// TIA Portal V17 export
// export: Created 2025-05-22T06:02:00.7232443Z, ExportSetting WithDefaults, DisplayName Totally Integrated Automation Portal, DisplayVersion V17 Update 8, DisplayName TIA Portal Openness, DisplayVersion V17 Update 8, DisplayName TIA Portal Version Control Interface, DisplayVersion V17, DisplayName SINAMICS Startdrive Advanced, DisplayVersion V17 SP2, DisplayName SINAMICS Startdrive G110M, G120, G120C, G120D, G120P, G115D, DisplayVersion V17 SP2, DisplayName SINAMICS Startdrive G130, G150, S120, S150, SINAMICS MV, S210, DisplayVersion V17 SP2, DisplayName STEP 7 Professional, DisplayVersion V17 Update 8, DisplayName SINUMERIK ONE STEP 7 Toolbox, DisplayVersion V17 Update 12, DisplayName SINUMERIK ONE PLC Basic Program Plus, DisplayVersion V17 Update 12, DisplayName SINUMERIK 840D sl STEP 7 Toolbox, DisplayVersion V17 Update 12, DisplayName STEP 7 Safety, DisplayVersion V17 Update 6, DisplayName WinCC Advanced, DisplayVersion V17 Update 8
FUNCTION "FC17900_MAINTENANCE_SEQUENCE" : Void   // FC17001, LAD
{ S7_Optimized_Access := 'TRUE' }
VERSION : 0.1
// stored: AutoNumber false, IsIECCheckEnabled false, SetENOAutomatically false, UDAEnableTagReadback false
   VAR_INPUT
      START_REQ : Bool;
      NUMBER_STEPS : Int;
      FIRST_STEP_DONE : Bool;
      SECOND_STEP_DONE : Bool;
      THRID_STEP_DONE : Bool;
      FOURTH_STEP_DONE : Bool;
      FIFTH_STEP_DONE : Bool;
   END_VAR
   VAR_OUTPUT
      FIRST_OPERATOR_HELP : Bool;
      SECOND_OPERATOR_HELP : Bool;
      THRID_OPERATOR_HELP : Bool;
      FOURTH_OPERATOR_HELP : Bool;
      FIFTH_OPERATOR_HELP : Bool;
      MAINTENANCE_IN_PROGRESS : Bool;
   END_VAR
   VAR_TEMP
      OPTION_FIRST_STEP : Bool;
      OPTION_SECOND_STEP : Bool;
      OPTION_THRID_STEP : Bool;
      OPTION_FOURTH_STEP : Bool;
      OPTION_FIFTH_STEP : Bool;
      SEQUENCE : "SEQUENCE";
   END_VAR
   VAR_TEMP   // added for the SCL form of the ladder/FBD networks
      _w1 : Bool;
   END_VAR
BEGIN

REGION Network 1: RESET OPTIONS
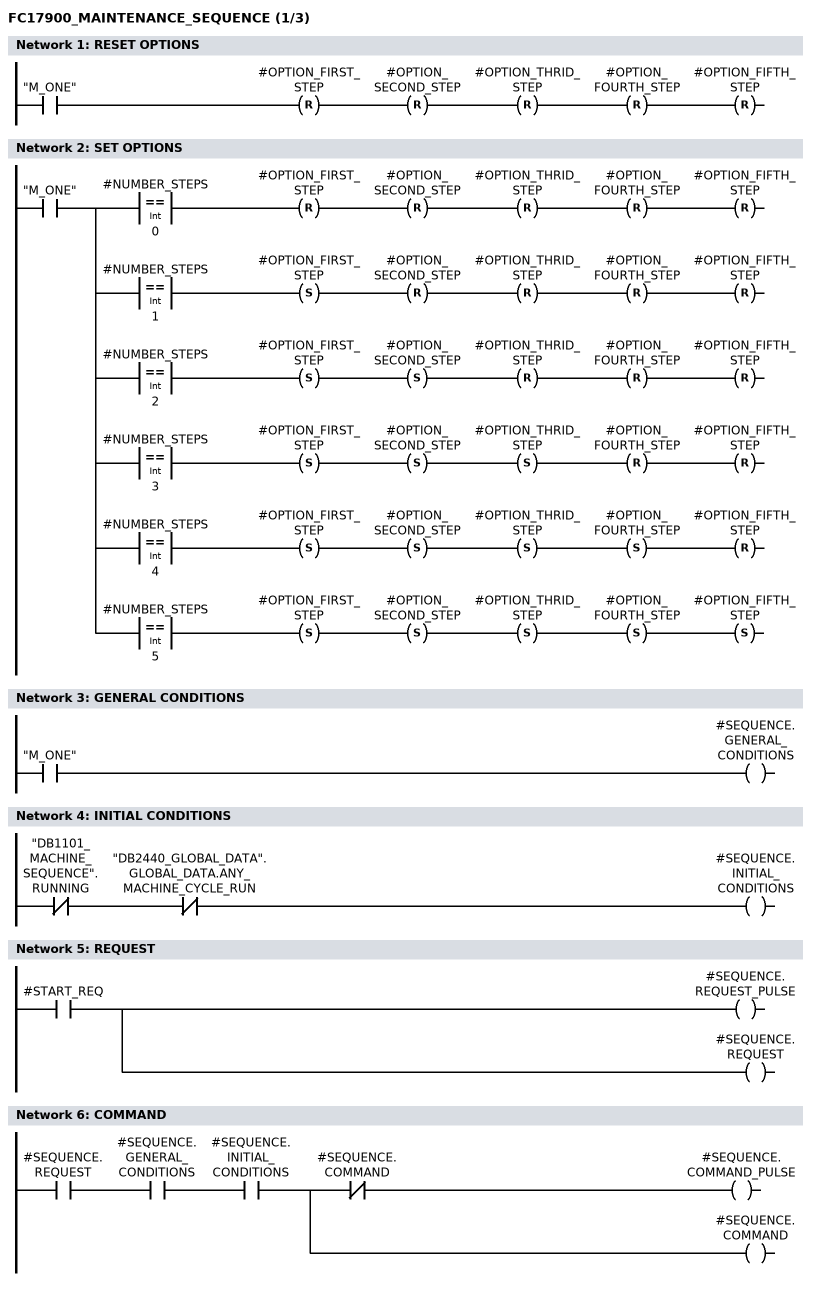
   RUNG wire#powerrail
      Contact( "M_ONE" )
      R_Coil( #OPTION_FIRST_STEP )
      R_Coil( #OPTION_SECOND_STEP )
      R_Coil( #OPTION_THRID_STEP )
      R_Coil( #OPTION_FOURTH_STEP )
      R_Coil( #OPTION_FIFTH_STEP )
   END_RUNG
   // the same network as SCL:
   IF "M_ONE" THEN
       #OPTION_FIRST_STEP := FALSE;
       #OPTION_SECOND_STEP := FALSE;
       #OPTION_THRID_STEP := FALSE;
       #OPTION_FOURTH_STEP := FALSE;
       #OPTION_FIFTH_STEP := FALSE;
   END_IF;
END_REGION

REGION Network 2: SET OPTIONS
   RUNG wire#powerrail
      Contact( "M_ONE" )
      wire#w1
      { S7_Templates := "SrcType := Int" } EQ_Contact(in1 := #NUMBER_STEPS, in2 := 0)
      R_Coil( #OPTION_FIRST_STEP )
      R_Coil( #OPTION_SECOND_STEP )
      R_Coil( #OPTION_THRID_STEP )
      R_Coil( #OPTION_FOURTH_STEP )
      R_Coil( #OPTION_FIFTH_STEP )
   END_RUNG
   RUNG wire#w1
      { S7_Templates := "SrcType := Int" } EQ_Contact(in1 := #NUMBER_STEPS, in2 := 1)
      S_Coil( #OPTION_FIRST_STEP )
      R_Coil( #OPTION_SECOND_STEP )
      R_Coil( #OPTION_THRID_STEP )
      R_Coil( #OPTION_FOURTH_STEP )
      R_Coil( #OPTION_FIFTH_STEP )
   END_RUNG
   RUNG wire#w1
      { S7_Templates := "SrcType := Int" } EQ_Contact(in1 := #NUMBER_STEPS, in2 := 2)
      S_Coil( #OPTION_FIRST_STEP )
      S_Coil( #OPTION_SECOND_STEP )
      R_Coil( #OPTION_THRID_STEP )
      R_Coil( #OPTION_FOURTH_STEP )
      R_Coil( #OPTION_FIFTH_STEP )
   END_RUNG
   RUNG wire#w1
      { S7_Templates := "SrcType := Int" } EQ_Contact(in1 := #NUMBER_STEPS, in2 := 3)
      S_Coil( #OPTION_FIRST_STEP )
      S_Coil( #OPTION_SECOND_STEP )
      S_Coil( #OPTION_THRID_STEP )
      R_Coil( #OPTION_FOURTH_STEP )
      R_Coil( #OPTION_FIFTH_STEP )
   END_RUNG
   RUNG wire#w1
      { S7_Templates := "SrcType := Int" } EQ_Contact(in1 := #NUMBER_STEPS, in2 := 4)
      S_Coil( #OPTION_FIRST_STEP )
      S_Coil( #OPTION_SECOND_STEP )
      S_Coil( #OPTION_THRID_STEP )
      S_Coil( #OPTION_FOURTH_STEP )
      R_Coil( #OPTION_FIFTH_STEP )
   END_RUNG
   RUNG wire#w1
      { S7_Templates := "SrcType := Int" } EQ_Contact(in1 := #NUMBER_STEPS, in2 := 5)
      S_Coil( #OPTION_FIRST_STEP )
      S_Coil( #OPTION_SECOND_STEP )
      S_Coil( #OPTION_THRID_STEP )
      S_Coil( #OPTION_FOURTH_STEP )
      S_Coil( #OPTION_FIFTH_STEP )
   END_RUNG
   // the same network as SCL:
   IF "M_ONE" AND (#NUMBER_STEPS = 0) THEN
       #OPTION_FIRST_STEP := FALSE;
       #OPTION_SECOND_STEP := FALSE;
       #OPTION_THRID_STEP := FALSE;
       #OPTION_FOURTH_STEP := FALSE;
       #OPTION_FIFTH_STEP := FALSE;
   END_IF;
   IF "M_ONE" AND (#NUMBER_STEPS = 1) THEN
       #OPTION_FIRST_STEP := TRUE;
       #OPTION_SECOND_STEP := FALSE;
       #OPTION_THRID_STEP := FALSE;
       #OPTION_FOURTH_STEP := FALSE;
       #OPTION_FIFTH_STEP := FALSE;
   END_IF;
   IF "M_ONE" AND (#NUMBER_STEPS = 2) THEN
       #OPTION_FIRST_STEP := TRUE;
       #OPTION_SECOND_STEP := TRUE;
       #OPTION_THRID_STEP := FALSE;
       #OPTION_FOURTH_STEP := FALSE;
       #OPTION_FIFTH_STEP := FALSE;
   END_IF;
   IF "M_ONE" AND (#NUMBER_STEPS = 3) THEN
       #OPTION_FIRST_STEP := TRUE;
       #OPTION_SECOND_STEP := TRUE;
       #OPTION_THRID_STEP := TRUE;
       #OPTION_FOURTH_STEP := FALSE;
       #OPTION_FIFTH_STEP := FALSE;
   END_IF;
   IF "M_ONE" AND (#NUMBER_STEPS = 4) THEN
       #OPTION_FIRST_STEP := TRUE;
       #OPTION_SECOND_STEP := TRUE;
       #OPTION_THRID_STEP := TRUE;
       #OPTION_FOURTH_STEP := TRUE;
       #OPTION_FIFTH_STEP := FALSE;
   END_IF;
   IF "M_ONE" AND (#NUMBER_STEPS = 5) THEN
       #OPTION_FIRST_STEP := TRUE;
       #OPTION_SECOND_STEP := TRUE;
       #OPTION_THRID_STEP := TRUE;
       #OPTION_FOURTH_STEP := TRUE;
       #OPTION_FIFTH_STEP := TRUE;
   END_IF;
END_REGION

REGION Network 3: GENERAL CONDITIONS
   RUNG wire#powerrail
      Contact( "M_ONE" )
      Coil( #SEQUENCE.GENERAL_CONDITIONS )
   END_RUNG
   // the same network as SCL:
   #SEQUENCE.GENERAL_CONDITIONS := "M_ONE";
END_REGION

REGION Network 4: INITIAL CONDITIONS
   RUNG wire#powerrail
      I_Contact( "DB1101_MACHINE_SEQUENCE".RUNNING )
      I_Contact( "DB2440_GLOBAL_DATA".GLOBAL_DATA.ANY_MACHINE_CYCLE_RUN )
      Coil( #SEQUENCE.INITIAL_CONDITIONS )
   END_RUNG
   // the same network as SCL:
   #SEQUENCE.INITIAL_CONDITIONS := NOT "DB1101_MACHINE_SEQUENCE".RUNNING AND NOT "DB2440_GLOBAL_DATA".GLOBAL_DATA.ANY_MACHINE_CYCLE_RUN;
END_REGION

REGION Network 5: REQUEST
   RUNG wire#powerrail
      Contact( #START_REQ )
      wire#w1
      Coil( #SEQUENCE.REQUEST_PULSE )
   END_RUNG
   RUNG wire#w1
      Coil( #SEQUENCE.REQUEST )
   END_RUNG
   // the same network as SCL:
   #SEQUENCE.REQUEST_PULSE := #START_REQ;
   #SEQUENCE.REQUEST := #START_REQ;
END_REGION

REGION Network 6: COMMAND
   RUNG wire#powerrail
      Contact( #SEQUENCE.REQUEST )
      Contact( #SEQUENCE.GENERAL_CONDITIONS )
      Contact( #SEQUENCE.INITIAL_CONDITIONS )
      wire#w1
      I_Contact( #SEQUENCE.COMMAND )
      Coil( #SEQUENCE.COMMAND_PULSE )
   END_RUNG
   RUNG wire#w1
      Coil( #SEQUENCE.COMMAND )
   END_RUNG
   // the same network as SCL:
   #_w1 := #SEQUENCE.REQUEST AND #SEQUENCE.GENERAL_CONDITIONS AND #SEQUENCE.INITIAL_CONDITIONS;
   #SEQUENCE.COMMAND_PULSE := #_w1 AND NOT #SEQUENCE.COMMAND;
   #SEQUENCE.COMMAND := #_w1;
END_REGION

REGION Network 7: RESET PLC AND CNC
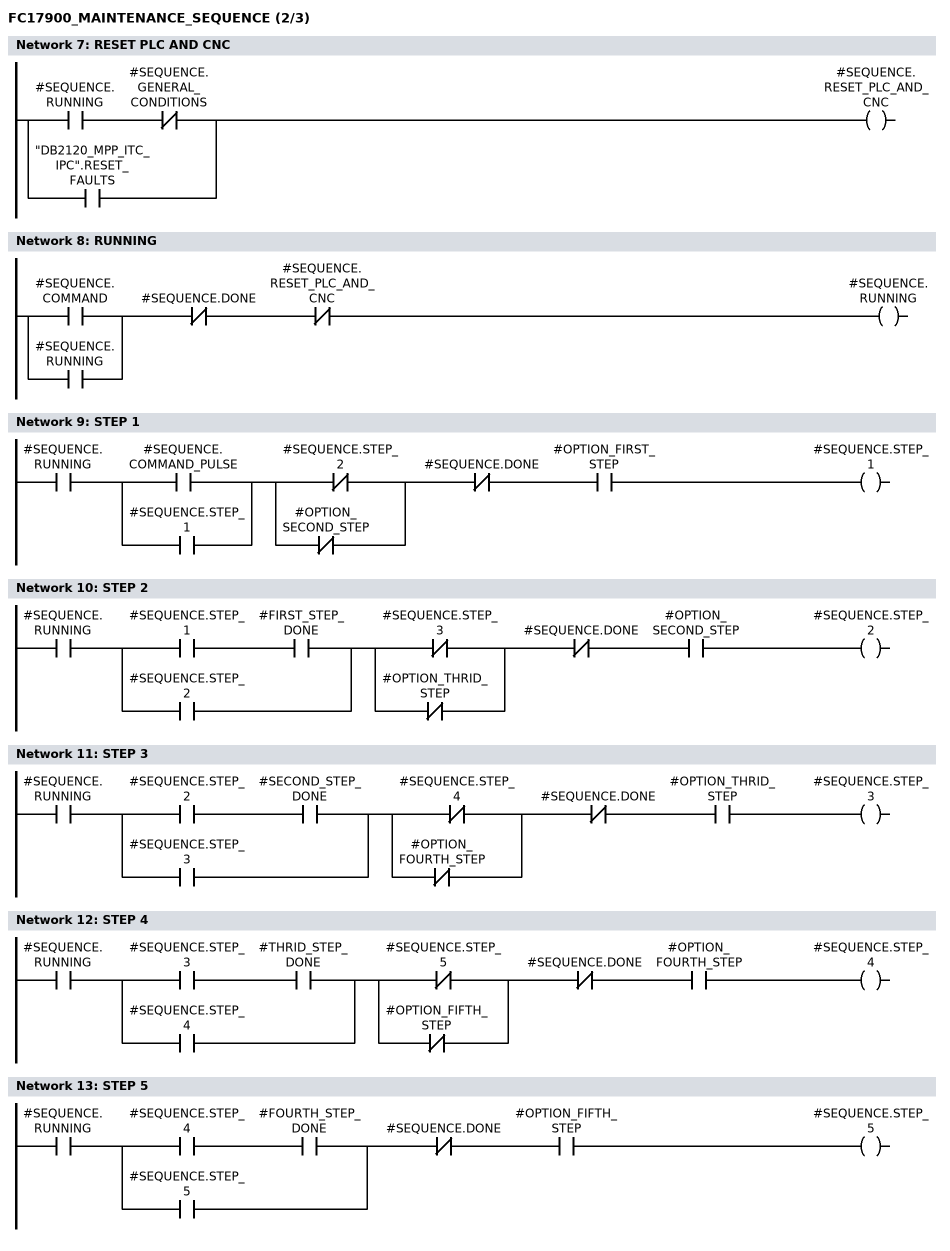
   RUNG wire#powerrail
      Contact( #SEQUENCE.RUNNING )
      I_Contact( #SEQUENCE.GENERAL_CONDITIONS )
      wire#w1
      Coil( #SEQUENCE.RESET_PLC_AND_CNC )
   END_RUNG
   RUNG wire#powerrail
      Contact( "DB2120_MPP_ITC_IPC".RESET_FAULTS )
   END_RUNG wire#w1
   // the same network as SCL:
   #SEQUENCE.RESET_PLC_AND_CNC := (#SEQUENCE.RUNNING AND NOT #SEQUENCE.GENERAL_CONDITIONS) OR "DB2120_MPP_ITC_IPC".RESET_FAULTS;
END_REGION

REGION Network 8: RUNNING
   RUNG wire#powerrail
      Contact( #SEQUENCE.COMMAND )
      wire#w1
      I_Contact( #SEQUENCE.DONE )
      I_Contact( #SEQUENCE.RESET_PLC_AND_CNC )
      Coil( #SEQUENCE.RUNNING )
   END_RUNG
   RUNG wire#powerrail
      Contact( #SEQUENCE.RUNNING )
   END_RUNG wire#w1
   // the same network as SCL:
   #SEQUENCE.RUNNING := (#SEQUENCE.COMMAND OR #SEQUENCE.RUNNING) AND NOT #SEQUENCE.DONE AND NOT #SEQUENCE.RESET_PLC_AND_CNC;
END_REGION

REGION Network 9: STEP 1
   RUNG wire#powerrail
      Contact( #SEQUENCE.RUNNING )
      wire#w1
      Contact( #SEQUENCE.COMMAND_PULSE )
      wire#w2
      I_Contact( #SEQUENCE.STEP_2 )
      wire#w3
      I_Contact( #SEQUENCE.DONE )
      Contact( #OPTION_FIRST_STEP )
      Coil( #SEQUENCE.STEP_1 )
   END_RUNG
   RUNG wire#w1
      Contact( #SEQUENCE.STEP_1 )
   END_RUNG wire#w2
   RUNG wire#w2
      I_Contact( #OPTION_SECOND_STEP )
   END_RUNG wire#w3
   // the same network as SCL:
   #SEQUENCE.STEP_1 := #SEQUENCE.RUNNING AND (#SEQUENCE.COMMAND_PULSE OR #SEQUENCE.STEP_1) AND (NOT #SEQUENCE.STEP_2 OR NOT #OPTION_SECOND_STEP) AND NOT #SEQUENCE.DONE AND #OPTION_FIRST_STEP;
END_REGION

REGION Network 10: STEP 2
   RUNG wire#powerrail
      Contact( #SEQUENCE.RUNNING )
      wire#w1
      Contact( #SEQUENCE.STEP_1 )
      Contact( #FIRST_STEP_DONE )
      wire#w2
      I_Contact( #SEQUENCE.STEP_3 )
      wire#w3
      I_Contact( #SEQUENCE.DONE )
      Contact( #OPTION_SECOND_STEP )
      Coil( #SEQUENCE.STEP_2 )
   END_RUNG
   RUNG wire#w1
      Contact( #SEQUENCE.STEP_2 )
   END_RUNG wire#w2
   RUNG wire#w2
      I_Contact( #OPTION_THRID_STEP )
   END_RUNG wire#w3
   // the same network as SCL:
   #SEQUENCE.STEP_2 := #SEQUENCE.RUNNING AND ((#SEQUENCE.STEP_1 AND #FIRST_STEP_DONE) OR #SEQUENCE.STEP_2) AND (NOT #SEQUENCE.STEP_3 OR NOT #OPTION_THRID_STEP) AND NOT #SEQUENCE.DONE AND #OPTION_SECOND_STEP;
END_REGION

REGION Network 11: STEP 3
   RUNG wire#powerrail
      Contact( #SEQUENCE.RUNNING )
      wire#w1
      Contact( #SEQUENCE.STEP_2 )
      Contact( #SECOND_STEP_DONE )
      wire#w2
      I_Contact( #SEQUENCE.STEP_4 )
      wire#w3
      I_Contact( #SEQUENCE.DONE )
      Contact( #OPTION_THRID_STEP )
      Coil( #SEQUENCE.STEP_3 )
   END_RUNG
   RUNG wire#w1
      Contact( #SEQUENCE.STEP_3 )
   END_RUNG wire#w2
   RUNG wire#w2
      I_Contact( #OPTION_FOURTH_STEP )
   END_RUNG wire#w3
   // the same network as SCL:
   #SEQUENCE.STEP_3 := #SEQUENCE.RUNNING AND ((#SEQUENCE.STEP_2 AND #SECOND_STEP_DONE) OR #SEQUENCE.STEP_3) AND (NOT #SEQUENCE.STEP_4 OR NOT #OPTION_FOURTH_STEP) AND NOT #SEQUENCE.DONE AND #OPTION_THRID_STEP;
END_REGION

REGION Network 12: STEP 4
   RUNG wire#powerrail
      Contact( #SEQUENCE.RUNNING )
      wire#w1
      Contact( #SEQUENCE.STEP_3 )
      Contact( #THRID_STEP_DONE )
      wire#w2
      I_Contact( #SEQUENCE.STEP_5 )
      wire#w3
      I_Contact( #SEQUENCE.DONE )
      Contact( #OPTION_FOURTH_STEP )
      Coil( #SEQUENCE.STEP_4 )
   END_RUNG
   RUNG wire#w1
      Contact( #SEQUENCE.STEP_4 )
   END_RUNG wire#w2
   RUNG wire#w2
      I_Contact( #OPTION_FIFTH_STEP )
   END_RUNG wire#w3
   // the same network as SCL:
   #SEQUENCE.STEP_4 := #SEQUENCE.RUNNING AND ((#SEQUENCE.STEP_3 AND #THRID_STEP_DONE) OR #SEQUENCE.STEP_4) AND (NOT #SEQUENCE.STEP_5 OR NOT #OPTION_FIFTH_STEP) AND NOT #SEQUENCE.DONE AND #OPTION_FOURTH_STEP;
END_REGION

REGION Network 13: STEP 5
   RUNG wire#powerrail
      Contact( #SEQUENCE.RUNNING )
      wire#w1
      Contact( #SEQUENCE.STEP_4 )
      Contact( #FOURTH_STEP_DONE )
      wire#w2
      I_Contact( #SEQUENCE.DONE )
      Contact( #OPTION_FIFTH_STEP )
      Coil( #SEQUENCE.STEP_5 )
   END_RUNG
   RUNG wire#w1
      Contact( #SEQUENCE.STEP_5 )
   END_RUNG wire#w2
   // the same network as SCL:
   #SEQUENCE.STEP_5 := #SEQUENCE.RUNNING AND ((#SEQUENCE.STEP_4 AND #FOURTH_STEP_DONE) OR #SEQUENCE.STEP_5) AND NOT #SEQUENCE.DONE AND #OPTION_FIFTH_STEP;
END_REGION

REGION Network 14: DONE
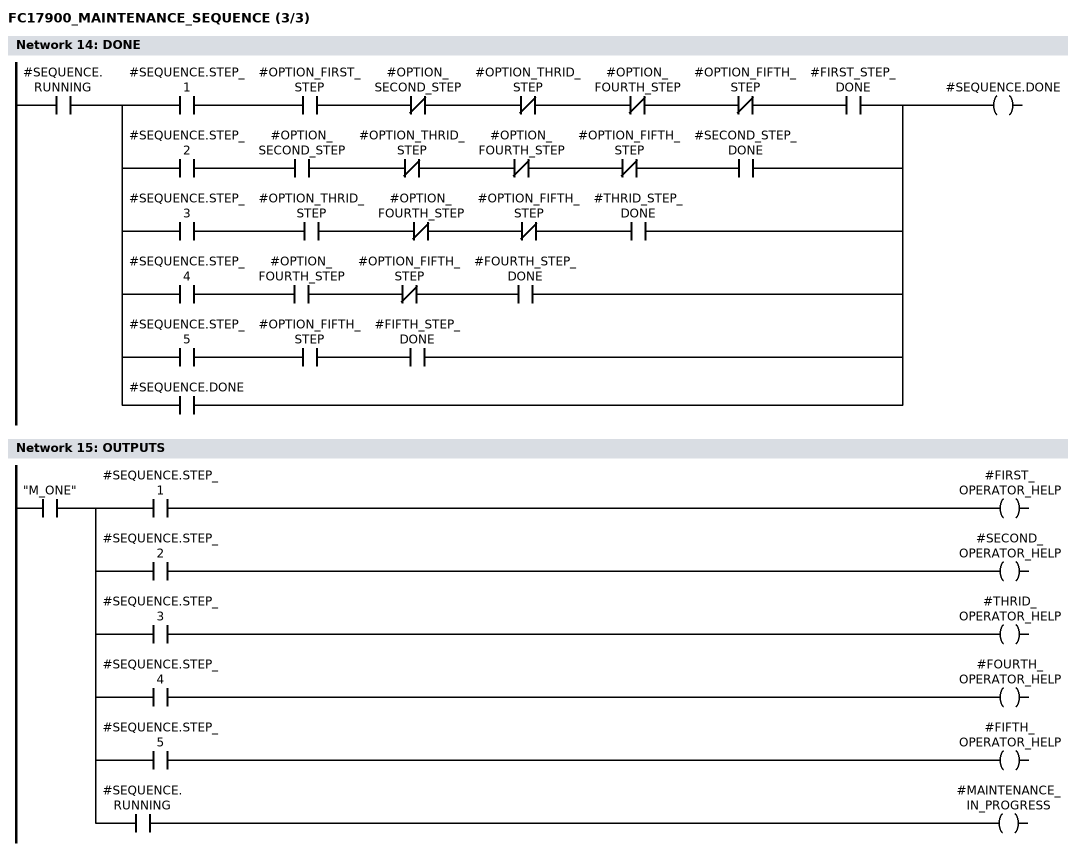
   RUNG wire#powerrail
      Contact( #SEQUENCE.RUNNING )
      wire#w1
      Contact( #SEQUENCE.STEP_1 )
      Contact( #OPTION_FIRST_STEP )
      I_Contact( #OPTION_SECOND_STEP )
      I_Contact( #OPTION_THRID_STEP )
      I_Contact( #OPTION_FOURTH_STEP )
      I_Contact( #OPTION_FIFTH_STEP )
      Contact( #FIRST_STEP_DONE )
      wire#w2
      Coil( #SEQUENCE.DONE )
   END_RUNG
   RUNG wire#w1
      Contact( #SEQUENCE.STEP_2 )
      Contact( #OPTION_SECOND_STEP )
      I_Contact( #OPTION_THRID_STEP )
      I_Contact( #OPTION_FOURTH_STEP )
      I_Contact( #OPTION_FIFTH_STEP )
      Contact( #SECOND_STEP_DONE )
   END_RUNG wire#w2
   RUNG wire#w1
      Contact( #SEQUENCE.STEP_3 )
      Contact( #OPTION_THRID_STEP )
      I_Contact( #OPTION_FOURTH_STEP )
      I_Contact( #OPTION_FIFTH_STEP )
      Contact( #THRID_STEP_DONE )
   END_RUNG wire#w2
   RUNG wire#w1
      Contact( #SEQUENCE.STEP_4 )
      Contact( #OPTION_FOURTH_STEP )
      I_Contact( #OPTION_FIFTH_STEP )
      Contact( #FOURTH_STEP_DONE )
   END_RUNG wire#w2
   RUNG wire#w1
      Contact( #SEQUENCE.STEP_5 )
      Contact( #OPTION_FIFTH_STEP )
      Contact( #FIFTH_STEP_DONE )
   END_RUNG wire#w2
   RUNG wire#w1
      Contact( #SEQUENCE.DONE )
   END_RUNG wire#w2
   // the same network as SCL:
   #SEQUENCE.DONE := #SEQUENCE.RUNNING AND ((#SEQUENCE.STEP_1 AND #OPTION_FIRST_STEP AND NOT #OPTION_SECOND_STEP AND NOT #OPTION_THRID_STEP AND NOT #OPTION_FOURTH_STEP AND NOT #OPTION_FIFTH_STEP AND #FIRST_STEP_DONE) OR (#SEQUENCE.STEP_2 AND #OPTION_SECOND_STEP AND NOT #OPTION_THRID_STEP AND NOT #OPTION_FOURTH_STEP AND NOT #OPTION_FIFTH_STEP AND #SECOND_STEP_DONE) OR (#SEQUENCE.STEP_3 AND #OPTION_THRID_STEP AND NOT #OPTION_FOURTH_STEP AND NOT #OPTION_FIFTH_STEP AND #THRID_STEP_DONE) OR (#SEQUENCE.STEP_4 AND #OPTION_FOURTH_STEP AND NOT #OPTION_FIFTH_STEP AND #FOURTH_STEP_DONE) OR (#SEQUENCE.STEP_5 AND #OPTION_FIFTH_STEP AND #FIFTH_STEP_DONE) OR #SEQUENCE.DONE);
END_REGION

REGION Network 15: OUTPUTS
   RUNG wire#powerrail
      Contact( "M_ONE" )
      wire#w1
      Contact( #SEQUENCE.STEP_1 )
      Coil( #FIRST_OPERATOR_HELP )
   END_RUNG
   RUNG wire#w1
      Contact( #SEQUENCE.STEP_2 )
      Coil( #SECOND_OPERATOR_HELP )
   END_RUNG
   RUNG wire#w1
      Contact( #SEQUENCE.STEP_3 )
      Coil( #THRID_OPERATOR_HELP )
   END_RUNG
   RUNG wire#w1
      Contact( #SEQUENCE.STEP_4 )
      Coil( #FOURTH_OPERATOR_HELP )
   END_RUNG
   RUNG wire#w1
      Contact( #SEQUENCE.STEP_5 )
      Coil( #FIFTH_OPERATOR_HELP )
   END_RUNG
   RUNG wire#w1
      Contact( #SEQUENCE.RUNNING )
      Coil( #MAINTENANCE_IN_PROGRESS )
   END_RUNG
   // the same network as SCL:
   #FIRST_OPERATOR_HELP := "M_ONE" AND #SEQUENCE.STEP_1;
   #SECOND_OPERATOR_HELP := "M_ONE" AND #SEQUENCE.STEP_2;
   #THRID_OPERATOR_HELP := "M_ONE" AND #SEQUENCE.STEP_3;
   #FOURTH_OPERATOR_HELP := "M_ONE" AND #SEQUENCE.STEP_4;
   #FIFTH_OPERATOR_HELP := "M_ONE" AND #SEQUENCE.STEP_5;
   #MAINTENANCE_IN_PROGRESS := "M_ONE" AND #SEQUENCE.RUNNING;
END_REGION
END_FUNCTION
